FUNCTION_BLOCK CbVtStatus (* This function is called in case of every page change - you can do e. g. initialisations ... *)
  (* Standard: ISO 11783-6; Description: Copyright (c) 2022 HR Agrartechnik GmbH This program and the accompanying materials are made available under the terms of the Eclipse Public License 2.0 which is available at https://www.eclipse.org/legal/epl-2.0/ SPDX-License-Identifier: EPL-2.0 This function is called in case of every page change - you can do e. g. initialisations ... *)
  (* Version 1.2, 2026-09-05, Franz Höpfinger, HR Agrartechnik GmbH, Populate SCALING-TEST status outputs *)
  (* Version 1.1, 2026-09-05, Franz Höpfinger, HR Agrartechnik GmbH, Added SCALING-TEST status outputs (wSKM_Scal, w_DMScal, u8SKM_Number, qScalingTestEnabled) *)
  (* Version 1.0, 2022-07-20, Franz Höpfinger, HR Agrartechnik GmbH *)
  PACKAGE isobus::UT::status;
  IMPORT isobus::UT::Q::const::IDs::ID_NULL;
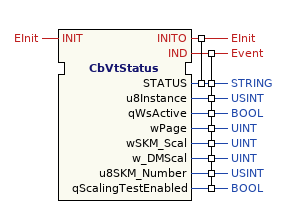
  EVENT_INPUT
    INIT : EInit; (* Service Initialization *)
  END_EVENT
  EVENT_OUTPUT
    INITO : EInit WITH STATUS; (* Initialization Confirm *)
    IND WITH STATUS, wPage, qWsActive, u8Instance, wSKM_Scal, w_DMScal, u8SKM_Number, qScalingTestEnabled; (* Indication from Resource *)
  END_EVENT
  VAR_OUTPUT
    STATUS : STRING; (* Service Status *)
    u8Instance : USINT; (* Identifier of the client instance *)
    qWsActive : BOOL; (* true, if the working set is active (displayed on screen) *)
    wPage : UINT := ID_NULL; (* Contains the object ID of the open/last mask, or NULL object ID if unknown (ID_NULL = 0xFFFF) *)
    wSKM_Scal : UINT; (* Softkey Mask scaling factor (PoolSoftKeyMaskScalFaktor), unit 1/10000 (10000 = 100%) - possibly overridden by SCALING-TEST *)
    w_DMScal : UINT; (* Data Mask scaling factor (PoolDataMaskScalFaktor), unit 1/10000 (10000 = 100%) - possibly overridden by SCALING-TEST *)
    u8SKM_Number : USINT; (* Number of physical softkeys (VT_PHYSICALSOFTKEYS/sknu), valid range 6..11 - possibly overridden by SCALING-TEST *)
    qScalingTestEnabled : BOOL; (* true if the SCALING-TEST override ([ScalingTest] enable=1 in settings.ini) is active *)
  END_VAR
END_FUNCTION_BLOCK
